ABB RobotStudio station: EGM.rsstnx

Station EGM (saved by RobotStudio 25.1.11133.0)
Controller CRB15000_5_95
  mechanical unit ROB_1: CRB15000_5_95__02, 6 joints, base frame (0, 0, 0) mm
Layout (positions relative to the parent item):
  - CRB15000_5_95__02 [mechanism, from %ABB.RobotStudio.Models.CRB15000%\CRB15000_5_95__02.rslib] at (0, 0, 0) mm; joint values [0, -0.1417, 0.3789, 0, 1.3335, 0] (rad or m)
